FUNCTION_BLOCK Camera (* Service Interface Function Block Type *)
  (* Standard: 61499-2 *)
  (* Version 0.0, 2012-05-26, 4DIAC-IDE, 4DIAC-Consortium *)
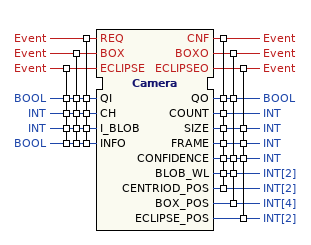
  EVENT_INPUT
    REQ WITH QI, CH, I_BLOB, INFO; (* track_update and returns all information *)
    BOX WITH I_BLOB, CH, QI, INFO;
    ECLIPSE WITH QI, CH, I_BLOB, INFO;
  END_EVENT
  EVENT_OUTPUT
    CNF WITH QO, COUNT, SIZE, FRAME, CENTRIOD_POS, CONFIDENCE, BLOB_WL; (* CENTRIOD Confirmation of Requested Service *)
    BOXO WITH CONFIDENCE, BLOB_WL, QO, BOX_POS;
    ECLIPSEO WITH ECLIPSE_POS, CONFIDENCE, FRAME, SIZE;
  END_EVENT
  VAR_INPUT
    QI : BOOL; (* Event Input Qualifier *)
    CH : INT; (* channel (0-3) of blob *)
    I_BLOB : INT; (* index of Blob, where 0 is the largest and default, Up to 9 blobs channels supported *)
    INFO : BOOL; (* prints outputs if true=1 *)
  END_VAR
  VAR_OUTPUT
    QO : BOOL; (* Event Output Qualifier *)
    COUNT : INT; (* Number of blobs on a channel. *)
    SIZE : INT; (* size of blob from channel CH and INDEX in pixels *)
    FRAME : INT; (* frame number used to generate the tracking data *)
    CONFIDENCE : INT; (* % confidence for seeing the blob in pixel area/bounding box area for CH/INDEX *)
    BLOB_WL : ARRAY [0..1] OF INT; (* [Width x,Length y] in pixel  of the bounding box for the blob from CH/INDEX *)
    CENTRIOD_POS : ARRAY [0..1] OF INT; (* [X,Y] pixel [x,y] coordinate of the centroid for the blob *)
    BOX_POS : ARRAY [0..3] OF INT; (* [RT,LT,TOP,BOTTOM] of blob box *)
    ECLIPSE_POS : ARRAY [0..1] OF INT; (* [MAJOR, MINOR] length in pixels of the axis of the bounding ECLIPSE for the blob *)
  END_VAR
  SERVICE APPLICATION/RESOURCE (* Service Interface Function Block Type *)
    SEQUENCE normal_establishment
      APPLICATION.INIT+(PARAMS) -> APPLICATION.INITO+(PARAMS);
    END_SEQUENCE
    SEQUENCE unsuccessful_establishment
      APPLICATION.INIT+(PARAMS) -> APPLICATION.INITO-(STATUS);
    END_SEQUENCE
    SEQUENCE request_confirm
      APPLICATION.REQ+(SD) -> APPLICATION.CNF+(RD);
    END_SEQUENCE
    SEQUENCE request_inhibited
      APPLICATION.REQ-(SD) -> APPLICATION.CNF-(STATUS);
    END_SEQUENCE
    SEQUENCE request_error
      APPLICATION.REQ+(SD) -> APPLICATION.CNF-(STATUS);
    END_SEQUENCE
    SEQUENCE indication_response
      RESOURCE.indicate(RD) -> APPLICATION.IND+(RD);
      APPLICATION.RSP(QI,SD) -> RESOURCE.response(QI,SD);
    END_SEQUENCE
    SEQUENCE indication_inhibited
      RESOURCE.indicate(RD,QI=FALSE) -> RESOURCE.inhibited();
    END_SEQUENCE
    SEQUENCE error_indication
      RESOURCE.error(STATUS) -> APPLICATION.IND-(STATUS);
    END_SEQUENCE
    SEQUENCE application_initiated_termination
      APPLICATION.INIT-() -> APPLICATION.INITO-(STATUS);
    END_SEQUENCE
    SEQUENCE resource_initiated_termination
      -> APPLICATION.INITO-(STATUS);
    END_SEQUENCE
  END_SERVICE
END_FUNCTION_BLOCK
